PROGRAM P_Demo_FB_DMXGetDeviceModelDescription
VAR
    fbGetModelDesc    : FB_DMXGetDeviceModelDescription; // 读型号描述
    stDmxCmdBuffer    : ST_DMXCommandBuffer;          // 与通讯 FB 共用
    wTargetManufId    : WORD := 16#4241;              // 目标灯具厂商 ID
    dwTargetDeviceId  : DWORD := 16#12131415;         // 目标灯具设备 ID
    byTargetPort      : BYTE := 0;                    // 根设备通道 0
    bDoRead           : BOOL := FALSE;                // 在线给一次上升沿触发
    bBusy             : BOOL;
    bError            : BOOL;
    udiErrId          : UDINT;
    sModelDesc        : STRING;                       // 型号描述文本
END_VAR

// ============================================================
// Tc2_DMX.FB_DMXGetDeviceModelDescription 演示程序
// ============================================================
// 场景：资产盘点/备件管理：批量读出总线每盏灯的型号描述，自动生成设备清单便于采购备件。
// 价值：把型号信息从设备直接读出，资产清单与现场实物一致，免去人工抄录。
// 验证：给 bDoRead 一次上升沿 -> bBusy 短暂 TRUE -> 回 FALSE 后 sModelDesc 即厂商型号描述文本；不支持该 PID 的设备 bError 且 udiErrId=0x8010。
// 验证步骤：
//   1. 右键 PLC 项目下 POUs 文件夹 → Add → Existing Item → 选本 .TcPOU 文件
//   2. 引用 Tc2_DMX；同项目里放一个 FB_EL6851CommunicationEx 实例并共用 stDmxCmdBuffer（非 CycleMode）
//   3. 编译 → 登录 → 运行；按上方『验证』行在线给上升沿观察
// ============================================================

fbGetModelDesc(
    bStart                     := bDoRead,
    wDestinationManufacturerId := wTargetManufId,
    dwDestinationDeviceId      := dwTargetDeviceId,
    byPortId                   := byTargetPort,
    dwOptions                  := 0,
    stCommandBuffer            := stDmxCmdBuffer,
    bBusy                      => bBusy,
    bError                     => bError,
    udiErrorId                 => udiErrId,
    sDeviceModelDescription    => sModelDesc
);

END_PROGRAM

(* stored: Version 1.1.0.1, ProductVersion 3.1.4024.5
   POU P_Demo_FB_DMXGetDeviceModelDescription: Id {7f24ba09-e867-5b58-a8f0-697599ef1c7a}, SpecialFunc None *)
